///EL2032 | 2-channel digital output terminal 24 V DC, 2 A, diagnostics
FUNCTION_BLOCK EL2032

VAR_INPUT
	En: BOOL;
	bDo_1: BOOL;
	bDo_2: BOOL;
	iTerminal_ID : INT;
	ErrorSystem : POINTER TO ST_ErrorSystem;
END_VAR

VAR_OUTPUT
	EnO: BOOL;
	bDiag_1: BOOL;
	bDiag_2: BOOL;
	bError: BOOL;
END_VAR

VAR
	Diag_1_Diag AT %I*: BOOL;
	Diag_2_Diag AT %I*: BOOL;
	Channel_1_Output AT %Q*: BOOL;
	Channel_2_Output AT %Q*: BOOL;
	WcState_WcState AT %I*: BOOL;
	InfoData_State AT %I*: UINT;
	
	//FB-s
	EL2032_Error : FB_TerminalError;
END_VAR

EnO:=En;

//Error FB instance
EL2032_Error(
	En := TRUE,
	iTerminal_ID := iTerminal_ID,
	bWcState := WcState_WcState,
	uiInfoData_State := InfoData_State,
	pErrorSystem := ErrorSystem,
	bError => bError,
);

IF En THEN
	IF bError=FALSE THEN
		bDiag_1:=Diag_1_Diag;
		bDiag_2:=Diag_2_Diag;
		Channel_1_Output:=bDo_1;
		Channel_2_Output:=bDo_2;
	ELSE
		bDiag_1:=FALSE;
		bDiag_2:=FALSE;
	END_IF
END_IF

END_FUNCTION_BLOCK

(* stored: Version 1.1.0.1, ProductVersion 3.1.4022.10
   POU EL2032: Id {246ebfd8-3ec9-476c-9b1f-49b7848e5eaf}, SpecialFunc None *)
